(* CODESYS project TAC_Events.library
   Author: Mit Patel
   Version: 0.1.1.2
   Description: V0.1.1.0 - Initial
      V0.1.1.1 - Create RPC Sink
      V0.1.1.2 - Separate Buffer and Sink Interfaces
   Title: TAC_Events
   DefaultNamespace: TAC_Events
   Placeholder: TAC_Events
   Company: Timberline Automation and Control Co.

Project tree, tasks and I/O mapping:
  libraries: Tc2_EtherCAT, * (Beckhoff Automation GmbH); Tc2_Standard, * (Beckhoff Automation GmbH); Tc2_System, * (Beckhoff Automation GmbH); Tc2_Utilities, * (Beckhoff Automation GmbH); Tc3_JsonXml, * (Beckhoff Automation GmbH)
  ImportUtilities/
    Logger/
      data type E_LogSeverity
      function F_LogDebug [ST]
      function F_LogError [ST]
      function F_Logger [ST]
      function F_LogInfo [ST]
      function F_LogWarning [ST]
      function block FB_LogErrorEdge [ST]
      function block FB_LogInfoEdge [ST]
      function block FB_LogOnEdge [ST]
      function block FB_LogWarningEdge [ST]
      interface I_ExternalLogger: AddToLog
    String/
      Large Concats/
        function F_ClearLarge [ST]
        function F_Concat3_Large [ST]
        function F_Concat4_Large [ST]
        function F_Concat5_Large [ST]
        function F_Concat6_Large [ST]
        function F_Concat7_Large [ST]
        function F_ConcatLarge [ST]
      function F_Concat3 [ST]
      function F_Concat4 [ST]
      function F_Concat5 [ST]
      function F_Concat6 [ST]
      function F_Concat7 [ST]
      function F_StringToTarg [ST]
      function F_TargToString [ST]
      data type LongString
    global variables LogConfig
  Library/
    EventLogger/
      Bases/
        function block T_InstanceNameBase [ST]: InstanceName, SetInstanceName
      EventBuffers/
        function block T_JsonEventBuffer [ST]: FindAvailableBuffer, FindOldestBuffer, ResetBuffer, AddEvent, GetEvents, Initialise, ConvertToJson, CopyJson, EndJson, StartJson
      EventSinks/
        function block FB_CsvFileEventSink [ST]: AddEvent, GetEvents, Initialise, CyclicLogic
        function block T_RpcEventSink [ST]: AddEvent, GetEvents, Initialise
      Functions/
        function F_GetLogSeverityFromTcEventSeverity [ST]
      Interfaces/
        interface I_EventBuffer: AddEvent, GetEvents, Initialise
        interface I_EventLogger: LogEvent, ShouldLogEvent
        interface I_EventSeverityHandler: ClearLocalSeverity, GetGlobalSeverity, GetLocalSeverity, SetGlobalSeverity, SetLocalSeverity
        interface I_EventSink: AddEvent, GetEvents, Initialise
        interface I_EventSinkHandler: AddSink, ClearSinks
        interface I_Logger: LogCritical, LogError, LogInfo, LogVerbose, LogWarning
      function block T_EventLogger [ST]: LogEvent, ShouldLogEvent, ClearLocalSeverity, GetGlobalSeverity, GetLocalSeverity, SetGlobalSeverity, SetLocalSeverity, AddSink, ClearSinks, LogCritical, LogError, LogInfo, LogVerbose, LogWarning
      function block T_Logger [ST]: LogEvent, ShouldLogEvent, ClearLocalSeverity, GetGlobalSeverity, GetLocalSeverity, SetGlobalSeverity, SetLocalSeverity, LogCritical, LogError, LogInfo, LogVerbose, LogWarning, FB_init
    GVLs/
      global variables Events
      global variables EventsConfig
    Structs/
      data type ST_EventMessageBuffer
      data type ST_EventMessageBufferPool
      data type ST_EventMessageParams
      data type T_BufferString
      data type T_MessageString
    Time/
      function block FB_UnixTimestamp [ST]: TimestampMs
      interface I_TimeProvider: TimestampMs
  Project Information/
    function F_GetCompany [ST]
    function F_GetTitle [ST]
    function F_GetVersion [ST]
  Version/
    global variables Global_Version
*)

// ImportUtilities/Logger/E_LogSeverity
{attribute 'qualified_only'}
TYPE
   E_LogSeverity :
   (
      Debug := 0,
      Info := ADSLOG_MSGTYPE_HINT,
      Warning := ADSLOG_MSGTYPE_WARN,
      Error := ADSLOG_MSGTYPE_ERROR,
      None := 1000
   ) DWORD;
END_TYPE

// ImportUtilities/String/LongString
TYPE
   LongString : STRING(StringsParams.MAX_STRING_LENGTH);
END_TYPE // use StringsParams.MAX_STRING_LENGTH to adjust length

// Library/Structs/ST_EventMessageBuffer
{attribute 'pack_mode' := '0'}
TYPE ST_EventMessageBuffer :
STRUCT
 	bufferIndex : UINT := 0;
	availableForWriting : BOOL := TRUE;
  count : UINT := 0;
  timestampMs : ULINT;
  
  bufferSize : UDINT := EventsConfig.MAX_BUFFER_SIZE;
  dataSize : UDINT := 0;
END_STRUCT
END_TYPE

// Library/Structs/ST_EventMessageBufferPool
{attribute 'pack_mode' := '0'}
TYPE ST_EventMessageBufferPool :
STRUCT
  bufferCount : UINT := EventsConfig.MAX_BUFFERS;
	currentDataBufferIndex : UINT := 0;
	dataBuffers : ARRAY [1..EventsConfig.MAX_BUFFERS] OF ST_EventMessageBuffer;
END_STRUCT
END_TYPE

// Library/Structs/ST_EventMessageParams
TYPE ST_EventMessageParams :
STRUCT	
  Severity : TcEventSeverity;
  Message : T_MessageString;
  Source : T_MaxString;
END_STRUCT
END_TYPE

// Library/Structs/T_BufferString
TYPE T_BufferString : STRING(EventsConfig.MAX_BUFFER_SIZE); END_TYPE

// Library/Structs/T_MessageString
TYPE T_MessageString : STRING(EventsConfig.MAX_LOG_MESSAGE_SIZE); END_TYPE

// ImportUtilities/LogConfig
{attribute 'qualified_only'}
VAR_GLOBAL
   // set level to log. Lower log level includes higher levels i.e. info does warning and Error. 
   LogLevel : E_LogSeverity := E_LogSeverity.None; // Turn messages off by default
   ExternalLogger : I_ExternalLogger; // permit logging to something else
END_VAR

// Library/GVLs/Events
{attribute 'qualified_only'}
VAR_GLOBAL CONSTANT
  {attribute 'hide'}
  {warning disable C0228}
  _eventLogger  : T_EventLogger;                      // Global instance of event logger which will log to all sinks.
  {warning restore C0228}

  EventLogger   : I_Logger := _eventLogger;           // Global accessor for logging events.
  EventSinks    : I_EventSinkHandler := _eventLogger; // Global accessor for adding/ resetting sinks.
END_VAR

// Library/GVLs/EventsConfig
{attribute 'qualified_only'}
// Buffer Config
VAR_GLOBAL CONSTANT
  MAX_BUFFERS : UINT := 4;                    // Number of buffers.
  MAX_BUFFER_SIZE : UDINT := 65535;           // Max size in bytes of a buffer.
  CYCLE_BUFFERS : BOOL := TRUE;               // Overwrite buffers when all buffers are full.
  MAX_LOG_MESSAGE_SIZE : UINT := 512;         // Max length of log message.
  
  CSV_LOG_FILE_NAME : T_MaxString := 'logs';      // Name for CSV log files. Will have the date appended (e.g. logs_2024_05_26).
  CSV_LOG_FILE_PATH : T_MaxString := '/var/log/'; // The path for log files if using FB_CsvFileEventSink.
END_VAR

// Logs config
VAR_GLOBAL CONSTANT
  MAX_SINKS : UINT := 4; // Number of sinks.
END_VAR

// Version/Global_Version
{attribute 'TcGenerated'}
{attribute 'no-analysis'}
{attribute 'linkalways'}
// This function has been automatically generated from the project information.
VAR_GLOBAL CONSTANT
	{attribute 'const_non_replaced'}
	stLibVersion_TAC_Events : ST_LibVersion := (iMajor := 0, iMinor := 1, iBuild := 1, iRevision := 2, nFlags := 0, sVersion := '0.1.1.2');
END_VAR

// ImportUtilities/Logger/F_LogDebug
FUNCTION F_LogDebug : STRING;
VAR_INPUT
   Message : T_MaxString;
END_VAR

F_LogDebug :=
   F_Logger(
      E_LogSeverity.Debug,
      CONCAT('DEBUG ', Message)
   );

END_FUNCTION

// ImportUtilities/Logger/F_Logger
FUNCTION F_Logger : STRING;
VAR_INPUT
   LogSeverity : E_LogSeverity;
   Message : T_MaxString;
END_VAR

IF (LogSeverity < E_LogSeverity.None)
   AND_THEN (LogSeverity >= LogConfig.LogLevel) THEN

   ADSLOGSTR(LogSeverity OR ADSLOG_MSGTYPE_LOG, Message, '');
   F_Logger := Message;

   IF LogConfig.ExternalLogger <> 0 THEN
      LogConfig.ExternalLogger.AddToLog(Message, LogSeverity);
   END_IF

END_IF

END_FUNCTION

// ImportUtilities/Logger/F_LogError
FUNCTION F_LogError : STRING;
VAR_INPUT
   Message : T_MaxString;
END_VAR

F_LogError := F_Logger(ADSLOG_MSGTYPE_ERROR, Message);

END_FUNCTION

// ImportUtilities/Logger/F_LogInfo
FUNCTION F_LogInfo : STRING;
VAR_INPUT
   Message : T_MaxString;
END_VAR

F_LogInfo := F_Logger(ADSLOG_MSGTYPE_HINT, Message);

END_FUNCTION

// ImportUtilities/Logger/F_LogWarning
FUNCTION F_LogWarning : STRING;
VAR_INPUT
   Message : T_MaxString;
END_VAR

F_LogWarning := F_Logger(ADSLOG_MSGTYPE_WARN, Message);

END_FUNCTION

// ImportUtilities/Logger/FB_LogErrorEdge
FUNCTION_BLOCK FB_LogErrorEdge
VAR_INPUT
   Event : BOOL; // Event flag
   Message : T_MaxString; // Log message
   EventFallingEdge : BOOL := FALSE; // Defined which edge: FALSE = rising TRUE = falling, 
END_VAR
VAR_OUTPUT
   Q : BOOL;
END_VAR
VAR
   fbLogEdge : FB_LogOnEdge;
END_VAR

fbLogEdge(
   Event := Event,
   Message := Message,
   LogSeverity := E_LogSeverity.Error,
   EventFallingEdge := EventFallingEdge,
   Q => Q
);

END_FUNCTION_BLOCK

// ImportUtilities/Logger/FB_LogOnEdge
FUNCTION_BLOCK FB_LogOnEdge
VAR_INPUT
   Event : BOOL; // look for edge here to log.
   Message : T_MaxString; // message
   LogSeverity : E_LogSeverity; // severity
   EventFallingEdge : BOOL := FALSE; // TRUE for falling edge, FALSE for rising edge.
END_VAR
VAR_OUTPUT
   Q : BOOL;
END_VAR
VAR
   rt : R_TRIG;
   ft : F_TRIG;
END_VAR
VAR_TEMP
   logNow : BOOL;
END_VAR

rt(CLK := Event);
ft(CLK := Event);

Q := SEL(EventFallingEdge, rt.Q, ft.Q);

IF Q THEN

   CASE LogSeverity OF

      E_LogSeverity.Info:
         F_LogInfo(Message);

      E_LogSeverity.Warning:
         F_LogWarning(Message);

      E_LogSeverity.Error:
         F_LogError(Message);
   ELSE

      F_LogError(
         CONCAT(
            'Error in FB_LogOnEdge, Logseverity incorrect. Log Message for event is : ',
            Message
         )
      );

   END_CASE

END_IF

END_FUNCTION_BLOCK

// ImportUtilities/Logger/FB_LogInfoEdge
FUNCTION_BLOCK FB_LogInfoEdge
VAR_INPUT
   Event : BOOL; // Event flag
   Message : T_MaxString; // Log message
   EventFallingEdge : BOOL := FALSE; // Defined which edge: FALSE = rising TRUE = falling, 
END_VAR
VAR_OUTPUT
   Q : BOOL;
END_VAR
VAR
   fbLogEdge : FB_LogOnEdge;
END_VAR

fbLogEdge(
   Event := Event,
   Message := Message,
   LogSeverity := E_LogSeverity.Info,
   EventFallingEdge := EventFallingEdge,
   Q => Q
);

END_FUNCTION_BLOCK

// ImportUtilities/Logger/FB_LogWarningEdge
FUNCTION_BLOCK FB_LogWarningEdge
VAR_INPUT
   Event : BOOL; // Event flag
   Message : T_MaxString; // Log message
   EventFallingEdge : BOOL := FALSE; // Defined which edge: FALSE = rising TRUE = falling, 
END_VAR
VAR_OUTPUT
   Q : BOOL;
END_VAR
VAR
   fbLogEdge : FB_LogOnEdge;
END_VAR

fbLogEdge(
   Event := Event,
   Message := Message,
   LogSeverity := E_LogSeverity.Warning,
   EventFallingEdge := EventFallingEdge,
   Q => Q
);

END_FUNCTION_BLOCK

// ImportUtilities/Logger/I_ExternalLogger
INTERFACE I_ExternalLogger

METHOD AddToLog
VAR_IN_OUT
   Message : T_MaxString;
END_VAR
VAR_INPUT
   LogSeverity : E_LogSeverity;
END_VAR
END_METHOD

END_INTERFACE

// ImportUtilities/String/Large Concats/F_ClearLarge
FUNCTION F_ClearLarge
VAR_IN_OUT CONSTANT
   stringToClear : LongString;
END_VAR

MEMSET(ADR(stringToClear), 16#0, sizeof(stringToClear));

END_FUNCTION

// ImportUtilities/String/Large Concats/F_Concat3_Large
FUNCTION F_Concat3_Large : LongString;
VAR_IN_OUT CONSTANT
   StringOne : LongString;
   StringTwo : LongString;
   StringThree : LongString;
END_VAR
VAR
   str : LongString;
END_VAR

str := F_ConcatLarge(StringTwo, StringThree);

F_Concat3_Large :=
   F_ConcatLarge(
      StringOne,
      str
   );

END_FUNCTION

// ImportUtilities/String/Large Concats/F_ConcatLarge
FUNCTION F_ConcatLarge : LongString
VAR_IN_OUT CONSTANT
   StringOne : LongString;
   StringTwo : LongString;
END_VAR
VAR
   i, sizeToCpy, teminatingCharPos, maxLen : DINT;
   response : LongString;
END_VAR

maxLen := TO_DINT(StringsParams.MAX_STRING_LENGTH) - 1; // - 1 allows for terminating character in last position.

IF LEN(stringOne) + LEN(StringTwo) > maxLen THEN
   sizeToCpy := maxLen - LEN(StringTwo); //need room for the terminating character
   teminatingCharPos := maxLen; // this is the index position for utf-8 string as byte array

ELSE
   sizeToCpy := LEN(StringOne);
   teminatingCharPos := LEN(StringOne) + LEN(StringTwo);

END_IF

// copy strings into response
MEMCPY(ADR(response), ADR(StringOne), TO_UDINT(sizeToCpy));
MEMCPY(ADR(response[sizeToCpy]), ADR(StringTwo), TO_UDINT(LEN(StringTwo)));

response[teminatingCharPos] := 16#0; // string terminating character
F_ConcatLarge := response;

END_FUNCTION

// ImportUtilities/String/Large Concats/F_Concat4_Large
FUNCTION F_Concat4_Large : LongString
VAR_IN_OUT CONSTANT
   sOne : LongString;
   sTwo : LongString;
   sThree : LongString;
   sFour : LongString;
END_VAR
VAR
   str : LongString;
END_VAR

str := F_Concat3_Large(sTwo, sThree, sFour);

F_Concat4_Large :=
   F_ConcatLarge(
      sOne,
      str
   );

END_FUNCTION

// ImportUtilities/String/Large Concats/F_Concat5_Large
FUNCTION F_Concat5_Large : LongString
VAR_IN_OUT CONSTANT
   sOne : LongString;
   sTwo : LongString;
   sThree : LongString;
   sFour : LongString;
   sFive : LongString;
END_VAR
VAR
   str : LongString;
END_VAR

str := F_Concat4_Large(sTwo, sThree, sFour, sFive);
F_Concat5_Large :=
   F_ConcatLarge(
      sOne,
      str
   );

END_FUNCTION

// ImportUtilities/String/Large Concats/F_Concat6_Large
FUNCTION F_Concat6_Large : LongString
VAR_IN_OUT CONSTANT
   sOne : LongString;
   sTwo : LongString;
   sThree : LongString;
   sFour : LongString;
   sFive : LongString;
   sSix : LongString;
END_VAR
VAR
   str : LongString;
END_VAR

str := F_Concat5_Large(sTwo, sThree, sFour, sFive, sSix);
F_Concat6_Large :=
   F_ConcatLarge(
      sOne,
      str
   );

END_FUNCTION

// ImportUtilities/String/Large Concats/F_Concat7_Large
FUNCTION F_Concat7_Large : LongString
VAR_IN_OUT CONSTANT
   sOne : LongString;
   sTwo : LongString;
   sThree : LongString;
   sFour : LongString;
   sFive : LongString;
   sSix : LongString;
   sSeven : LongString;
END_VAR
VAR
   str : LongString;
END_VAR

str := F_Concat6_Large(
   sTwo,
   sThree,
   sFour,
   sFive,
   sSix,
   sSeven
);

F_Concat7_Large :=
   F_ConcatLarge(
      sOne,
      str
   );

END_FUNCTION

// ImportUtilities/String/F_Concat3
FUNCTION F_Concat3 : T_MaxString
VAR_INPUT
   StringOne : STRING;
   StringTwo : STRING;
   StringThree : STRING;
END_VAR
VAR
   response : T_MaxString;
END_VAR

response := CONCAT(StringOne, StringTwo);
response := CONCAT(response, StringThree);
F_Concat3 := response;

END_FUNCTION

// ImportUtilities/String/F_Concat4
FUNCTION F_Concat4 : T_MaxString
VAR_INPUT
   sOne : STRING;
   sTwo : STRING;
   sThree : STRING;
   sFour : STRING;
END_VAR

F_Concat4 := CONCAT(
   sOne,
   F_Concat3(sTwo, sThree, sFour)
);

END_FUNCTION

// ImportUtilities/String/F_Concat5
FUNCTION F_Concat5 : T_MaxString
VAR_INPUT
   sOne : STRING;
   sTwo : STRING;
   sThree : STRING;
   sFour : STRING;
   sFive : STRING;
END_VAR

F_Concat5 := CONCAT(
   sOne,
   F_Concat4(sTwo, sThree, sFour, sFive)
);

END_FUNCTION

// ImportUtilities/String/F_Concat6
FUNCTION F_Concat6 : T_MaxString
VAR_INPUT
   sOne : STRING;
   sTwo : STRING;
   sThree : STRING;
   sFour : STRING;
   sFive : STRING;
   sSix : STRING;
END_VAR

F_Concat6 := CONCAT(
   sOne,
   F_Concat5(sTwo, sThree, sFour, sFive, sSix)
);

END_FUNCTION

// ImportUtilities/String/F_Concat7
FUNCTION F_Concat7 : T_MaxString
VAR_INPUT
   sOne : STRING;
   sTwo : STRING;
   sThree : STRING;
   sFour : STRING;
   sFive : STRING;
   sSix : STRING;
   sSeven : STRING;
END_VAR

F_Concat7 := CONCAT(
   sOne,
   F_Concat6(
      sTwo,
      sThree,
      sFour,
      sFive,
      sSix,
      sSeven
   )
);

END_FUNCTION

// ImportUtilities/String/F_StringToTarg
FUNCTION F_StringToTarg
VAR_INPUT
   StringToConvert : T_MaxString;
END_VAR
VAR_IN_OUT
   Targ : T_ARG;
END_VAR
VAR
   b : POINTER TO BOOL;
   b8 : POINTER TO BYTE;
   w : POINTER TO WORD;
   dw : POINTER TO DWORD;
   usi : POINTER TO USINT;
   si : POINTER TO SINT;
   ui : POINTER TO UINT;
   i : POINTER TO INT;
   udi : POINTER TO UDINT;
   di : POINTER TO DINT;
   str : POINTER TO STRING;
   re : POINTER TO REAL;
   lr : POINTER TO LREAL;
END_VAR

CASE Targ.eType OF

   E_ArgType.ARGTYPE_BOOL:
      b := Targ.pData;
      b^ := TO_BOOL(StringToConvert);

   E_ArgType.ARGTYPE_BYTE:
      b8 := Targ.pData;
      b8^ := TO_BYTE(StringToConvert);

   E_ArgType.ARGTYPE_WORD:
      w := Targ.pData;
      w^ := TO_WORD(StringToConvert);

   E_ArgType.ARGTYPE_DWORD:
      dw := Targ.pData;
      dw^ := TO_DWORD(StringToConvert);

   E_ArgType.ARGTYPE_USINT:
      usi := Targ.pData;
      usi^ := TO_USINT(StringToConvert);

   E_ArgType.ARGTYPE_SINT:
      si := Targ.pData;
      si^ := TO_SINT(StringToConvert);

   E_ArgType.ARGTYPE_UINT:
      ui := Targ.pData;
      ui^ := TO_UINT(StringToConvert);

   E_ArgType.ARGTYPE_INT:
      i := Targ.pData;
      i^ := TO_INT(StringToConvert);

   E_ArgType.ARGTYPE_UDINT:
      udi := Targ.pData;
      udi^ := TO_UDINT(StringToConvert);

   E_ArgType.ARGTYPE_DINT:
      di := Targ.pData;
      di^ := TO_DINT(StringToConvert);

   E_ArgType.ARGTYPE_STRING:
      str := Targ.pData;
      str^ := TO_STRING(StringToConvert);

   E_ArgType.ARGTYPE_REAL:
      re := Targ.pData;
      re^ := TO_REAL(StringToConvert);

   E_ArgType.ARGTYPE_LREAL:
      lr := Targ.pData;
      lr^ := TO_LREAL(StringToConvert);

ELSE
   F_LogWarning(
      CONCAT(
         'Unsupported type in Targ for string conversion: ',
         TO_STRING(Targ.eType)
      )
   );
END_CASE

END_FUNCTION

// ImportUtilities/String/F_TargToString
FUNCTION F_TargToString : T_MaxString
VAR_INPUT
   Targ : T_ARG;
END_VAR
VAR
   b : POINTER TO BOOL;
   b8 : POINTER TO BYTE;
   w : POINTER TO WORD;
   dw : POINTER TO DWORD;
   usi : POINTER TO USINT;
   si : POINTER TO SINT;
   ui : POINTER TO UINT;
   i : POINTER TO INT;
   udi : POINTER TO UDINT;
   di : POINTER TO DINT;
   str : POINTER TO STRING;
   re : POINTER TO REAL;
   lr : POINTER TO LREAL;
END_VAR

CASE Targ.eType OF

   E_ArgType.ARGTYPE_BOOL:
      b := Targ.pData;
      F_TargToString := TO_STRING(b^);

   E_ArgType.ARGTYPE_BYTE:
      b8 := Targ.pData;
      F_TargToString := TO_STRING(b8^);

   E_ArgType.ARGTYPE_WORD:
      w := Targ.pData;
      F_TargToString := TO_STRING(w^);

   E_ArgType.ARGTYPE_DWORD:
      dw := Targ.pData;
      F_TargToString := TO_STRING(dw^);

   E_ArgType.ARGTYPE_USINT:
      usi := Targ.pData;
      F_TargToString := TO_STRING(usi^);

   E_ArgType.ARGTYPE_SINT:
      si := Targ.pData;
      F_TargToString := TO_STRING(si^);

   E_ArgType.ARGTYPE_UINT:
      ui := Targ.pData;
      F_TargToString := TO_STRING(ui^);

   E_ArgType.ARGTYPE_INT:
      i := Targ.pData;
      F_TargToString := TO_STRING(i^);

   E_ArgType.ARGTYPE_UDINT:
      udi := Targ.pData;
      F_TargToString := TO_STRING(udi^);

   E_ArgType.ARGTYPE_DINT:
      di := Targ.pData;
      F_TargToString := TO_STRING(di^);

   E_ArgType.ARGTYPE_STRING:
      str := Targ.pData;
      F_TargToString := TO_STRING(str^);

   E_ArgType.ARGTYPE_REAL:
      re := Targ.pData;
      F_TargToString := TO_STRING(re^);

   E_ArgType.ARGTYPE_LREAL:
      lr := Targ.pData;
      F_TargToString := TO_STRING(lr^);

ELSE
   F_LogWarning(
      CONCAT(
         'Unsupported type in Targ for string conversion: ',
         TO_STRING(Targ.eType)
      )
   );
END_CASE

END_FUNCTION

// Library/EventLogger/Bases/T_InstanceNameBase
{attribute 'reflection'} 
FUNCTION_BLOCK PUBLIC T_InstanceNameBase
VAR
  {attribute 'instance-path'} 
  {attribute 'noinit'} 
  name : T_MaxString;
  
  _instanceName : T_MaxString;
  isInstanceNameSet : BOOL := FALSE;
END_VAR

PROPERTY FINAL InstanceName : T_MaxString; // returns the fully scoped variable name
GET
IF NOT isInstanceNameSet THEN
   setInstanceName();
END_IF

InstanceName := _instanceName;
END_GET
END_PROPERTY

METHOD PRIVATE SetInstanceName
VAR
	charsToDeleteFromPath : INT;
END_VAR
//Remove Solution_Name
charsToDeleteFromPath := FIND(name, '.');
_instanceName := DELETE(name, charsToDeleteFromPath, 1);
//Remove ProjectName
charsToDeleteFromPath := FIND(_instanceName, '.');
//gives us just "FirstDeclaredPOU.etc.etc..." from above.
_instanceName := DELETE(_instanceName, charsToDeleteFromPath, 1);
END_METHOD

END_FUNCTION_BLOCK

// Library/EventLogger/EventBuffers/T_JsonEventBuffer
// Event sink which buffers log messages/ events ready for polling via RPC calls to 'GetEvents'; a method of the I_EventSink interface. 
FUNCTION_BLOCK PUBLIC T_JsonEventBuffer EXTENDS T_InstanceNameBase IMPLEMENTS I_EventBuffer
VAR
  isInitialised : BOOL := FALSE;
  
  bufferPool : ST_EventMessageBufferPool;
  jWriters : ARRAY [1..EventsConfig.MAX_BUFFERS] OF FB_JsonSaxWriter;

  _timeProvider : I_TimeProvider := NULL;
  eventId : ULINT := 0;
END_VAR

VAR CONSTANT
  NULL : UDINT := 0;
END_VAR

// Finds the first available buffer, if unable to find one and CYCLE_BUFFERS is set to TRUE, then will search for the first oldest buffer based on its timestamp.
// With CYCLE_BUFFERS set to FALSE, events will be dropped.
// Returns the buffer index from the pool, 0 (invalid) if a buffer is not found.
METHOD PRIVATE FindAvailableBuffer : UINT
VAR
  iBuffer : UINT := 0;
  iAvailable : UINT := 0;
  iOldest : UINT := 0;
END_VAR
IF NOT isInitialised THEN
  F_LogWarning(CONCAT(InstanceName, ': Unable to FindAvailableBuffer. Sink is uninitialised.'));
  RETURN;
END_IF

iAvailable := 0;

FOR iBuffer := 1 TO EventsConfig.MAX_BUFFERS DO 
  IF bufferPool.dataBuffers[iBuffer].availableForWriting THEN
    iAvailable := iBuffer;
    EXIT;
	END_IF
END_FOR

IF EventsConfig.CYCLE_BUFFERS THEN
  // All buffers are full
  IF iAvailable = 0 THEN
    iOldest := FindOldestBuffer(FALSE);
    IF iOldest > 0 AND iOldest <= EventsConfig.MAX_BUFFERS THEN
      iAvailable := iOldest;
    END_IF
  END_IF
END_IF

FindAvailableBuffer := iAvailable;
END_METHOD

// Finds the oldest buffer in the pool and returns its buffer index. Will return 0 if unable to find an old buffer.
// If checkHasItems is set to TRUE, then will only search for buffers with items, otherwise all buffers in the pool are considered.
METHOD PRIVATE FindOldestBuffer : UINT
VAR_INPUT
  checkHasItems : BOOL := FALSE;
END_VAR

VAR
  iBuffer : UINT := 0;
  iOldest : UINT := 0;
  timeOldest : ULINT;
END_VAR
IF NOT isInitialised THEN
  F_LogWarning(CONCAT(InstanceName, ': Unable to FindOldestBuffer. Sink is uninitialised.'));
  RETURN;
END_IF

IF _timeProvider = NULL THEN
  F_LogWarning(CONCAT(InstanceName, ': Unable to FindOldestBuffer. _timeProvider is uninitialised.'));
  RETURN;
END_IF

timeOldest := _timeProvider.TimestampMs;
FOR iBuffer := 1 TO EventsConfig.MAX_BUFFERS DO
  IF bufferPool.dataBuffers[iBuffer].timestampMs < timeOldest THEN
    IF NOT checkHasItems OR_ELSE bufferPool.dataBuffers[iBuffer].count > 0 THEN
      timeOldest := bufferPool.dataBuffers[iBuffer].timestampMs;
      iOldest := iBuffer;
    END_IF
  END_IF
END_FOR
    
FindOldestBuffer := iOldest;
END_METHOD

// Resets a buffer based on the input buffer index and starts the buffer ready for new events to be added.
METHOD PRIVATE ResetBuffer
VAR_INPUT
  iBuffer : UINT := 0;
END_VAR
IF NOT isInitialised THEN
  F_LogWarning(CONCAT(InstanceName, ': Unable to ResetBuffer. Sink is uninitialised.'));
  RETURN;
END_IF

IF _timeProvider = NULL THEN
  F_LogWarning(CONCAT(InstanceName, ': Unable to ResetBuffer. _timeProvider is uninitialised.'));
  RETURN;
END_IF

IF iBuffer > 0 AND iBuffer <= EventsConfig.MAX_BUFFERS THEN
  StartJson(iBuffer);
  
  bufferPool.dataBuffers[iBuffer].bufferIndex := iBuffer;
  bufferPool.dataBuffers[iBuffer].availableForWriting := TRUE;
  bufferPool.dataBuffers[iBuffer].count := 0;
  bufferPool.dataBuffers[iBuffer].bufferSize := EventsConfig.MAX_BUFFER_SIZE;
  bufferPool.dataBuffers[iBuffer].dataSize := 0;
  
  bufferPool.dataBuffers[iBuffer].timestampMs := _timeProvider.TimestampMs;
END_IF
END_METHOD

// Adds an event to the buffer for later processing.
METHOD PUBLIC AddEvent
VAR_INPUT
  eventMessageParams : ST_EventMessageParams;
END_VAR

VAR
  totalSize, messageSize : UDINT := 0;
  buffer : REFERENCE TO ST_EventMessageBuffer := 0;
END_VAR

VAR_INST
  jWriterLocal : FB_JsonSaxWriter; // For calculating message size.
END_VAR

VAR CONSTANT
  END_JSON_ARRAY_SIZE : UINT := 3; // End array, end object and null terminator.
END_VAR
IF NOT isInitialised THEN
  F_LogWarning(CONCAT(InstanceName, ': Unable to AddEvent. Sink is uninitialised.'));
  RETURN;
END_IF

jWriterLocal.ResetDocument();
messageSize := ConvertToJson(eventMessageParams, jWriter := jWriterLocal);

IF bufferPool.currentDataBufferIndex = 0 OR bufferPool.currentDataBufferIndex > EventsConfig.MAX_BUFFERS THEN // Try to find an empty buffer.
	bufferPool.currentDataBufferIndex := FindAvailableBuffer();
  ResetBuffer(bufferPool.currentDataBufferIndex);
END_IF

IF bufferPool.currentDataBufferIndex > 0 AND bufferPool.currentDataBufferIndex <= EventsConfig.MAX_BUFFERS THEN 
  buffer REF= bufferPool.dataBuffers[bufferPool.currentDataBufferIndex];

  IF buffer.dataSize + messageSize > (EventsConfig.MAX_BUFFER_SIZE - END_JSON_ARRAY_SIZE) THEN  // Will adding this event cause the buffer to overflow?
    EndJson(bufferPool.currentDataBufferIndex);
    buffer.availableForWriting := FALSE; // Available for reading/ sending

	  bufferPool.currentDataBufferIndex := FindAvailableBuffer(); // Next buffer for writing. Will return 0 if no available buffers.
    ResetBuffer(bufferPool.currentDataBufferIndex);
  END_IF
END_IF

IF bufferPool.currentDataBufferIndex > 0 AND bufferPool.currentDataBufferIndex <= EventsConfig.MAX_BUFFERS THEN // Check bounds again due to buffer index change above.
  buffer REF= bufferPool.dataBuffers[bufferPool.currentDataBufferIndex]; // Buffer index has changed so update the internal ref.
  IF buffer.availableForWriting THEN
    ConvertToJson(eventMessageParams, jWriter := jWriters[bufferPool.currentDataBufferIndex]);
    totalSize := jWriters[bufferPool.currentDataBufferIndex].GetDocumentLength();                 
    buffer.dataSize := totalSize;
    buffer.count := buffer.count + 1;
    eventId := eventId + 1;
  END_IF
END_IF
END_METHOD

// Gets events currently stored in the buffer and copies them to the resultString, returning the total length of bytes copied.
METHOD PUBLIC GetEvents : UDINT
VAR_INPUT
  resultString : REFERENCE TO T_BufferString;
END_VAR

VAR
  iBuffer : UINT := 0;
  totalSize : UDINT := 0;
END_VAR

VAR CONSTANT
  // Note that the size returned from any 
  // json writer's GetDocumentLength method 
  // includes the null terminator, which we want to remove.
  // This is due to the JSON parsers in .NET or Influx's Telegraf, etc
  // not being able to understand the null terminator and throwing errors,
  // e.g. stating that there are additional characters at the end of the JSON payload.
  REMOVE_NULL_TERMINATOR : UDINT := 1;
END_VAR
IF NOT isInitialised THEN
  F_LogWarning(CONCAT(InstanceName, ': Unable to GetEvents. Sink is uninitialised.'));
  RETURN;
END_IF

iBuffer := FindOldestBuffer(TRUE);
IF iBuffer > 0 AND iBuffer <= EventsConfig.MAX_BUFFERS THEN
  IF NOT bufferPool.dataBuffers[iBuffer].availableForWriting THEN
    IF bufferPool.dataBuffers[iBuffer].count > 0 THEN
      totalSize := CopyJson(iBuffer, resultString);
      ResetBuffer(iBuffer);
    END_IF
  ELSE // Current buffer
    IF bufferPool.dataBuffers[iBuffer].count > 0 THEN
      bufferPool.dataBuffers[iBuffer].availableForWriting := FALSE; // Available for reading/ sending
      EndJson(iBuffer);
      totalSize := CopyJson(iBuffer, resultString);
      ResetBuffer(iBuffer);
      bufferPool.currentDataBufferIndex := FindAvailableBuffer(); // Next buffer for writing. Will return 0 if no available buffers.
      ResetBuffer(bufferPool.currentDataBufferIndex);
    END_IF
  END_IF
END_IF

GetEvents := totalSize - REMOVE_NULL_TERMINATOR;
END_METHOD

// Initialises the buffer including an I_TimeProvider for timestamping buffers and events.
METHOD PUBLIC Initialise
VAR_INPUT
	timeProvider : I_TimeProvider;
END_VAR

VAR
  iBuffer : UINT := 0;
END_VAR
_timeProvider := timeProvider;

IF _timeProvider = NULL THEN
  F_LogWarning(CONCAT(InstanceName, ': Unable to Initialise. _timeProvider is uninitialised.'));
  RETURN;
END_IF

isInitialised := TRUE;

FOR iBuffer := 1 TO EventsConfig.MAX_BUFFERS DO 
  ResetBuffer(iBuffer);
END_FOR
END_METHOD

// Converts the input eventMessageParams to JSON (without string copying).
METHOD PRIVATE ConvertToJson
VAR_INPUT
  eventMessageParams : ST_EventMessageParams;
END_VAR

VAR_OUTPUT
  docSize : UDINT;
END_VAR

VAR_IN_OUT
  jWriter : FB_JsonSaxWriter;
END_VAR

VAR
  timestampMs : ULINT;
  severity : T_MaxString;
END_VAR
IF NOT isInitialised THEN
  F_LogWarning(CONCAT(InstanceName, ': Unable to ConvertToJson. Sink is uninitialised.'));
  RETURN;
END_IF

IF _timeProvider = NULL THEN
  F_LogWarning(CONCAT(InstanceName, ': Unable to ConvertToJson. _timeProvider is uninitialised.'));
  RETURN;
END_IF

timestampMs := _timeProvider.TimestampMs;
severity := TO_STRING(eventMessageParams.Severity);

jWriter.StartObject();

  jWriter.AddKey('EventId');
  jWriter.AddUlint(eventId);

  jWriter.AddKeyString('Severity', severity);
  jWriter.AddKey('FileTime'); // Add unix timestamp
  jWriter.AddUlint(timestampMs);
  jWriter.AddKeyString('SourceName', eventMessageParams.Source); 
  jWriter.AddKeyString('MessageBody', eventMessageParams.Message);
  
jWriter.EndObject();

docSize := jWriter.GetDocumentLength();
END_METHOD

// Copies data in the JSON writer and returns the total length of bytes copied.
METHOD PRIVATE CopyJson : UDINT
VAR_INPUT
  iBuffer : UINT := 0;
  resultString : REFERENCE TO T_BufferString;
END_VAR

VAR
  totalSize : UDINT := 0;
END_VAR

VAR CONSTANT
  RESULT_STRING_SIZE : UDINT := SIZEOF(resultString);
END_VAR
IF NOT isInitialised THEN
  F_LogWarning(CONCAT(InstanceName, ': Unable to CopyJson. Sink is uninitialised.'));
  RETURN;
END_IF

IF iBuffer = 0 OR iBuffer > EventsConfig.MAX_BUFFERS THEN
	RETURN;
END_IF

MEMSET(ADR(resultString), 0, RESULT_STRING_SIZE); // Copy doc should overwrite resultString including null termination characters. 

totalSize := jWriters[iBuffer].CopyDocument
             (
               PDoc := resultString, 
               nDoc := RESULT_STRING_SIZE
             );
             
bufferPool.dataBuffers[iBuffer].dataSize := totalSize;
CopyJson := totalSize;
END_METHOD

// Ends the JSON string, ready for the JSON string to be copied.
METHOD PRIVATE EndJson
VAR_INPUT
  iBuffer : UINT := 0;
END_VAR
IF NOT isInitialised THEN
  F_LogWarning(CONCAT(InstanceName, ': Unable to EndJson. Sink is uninitialised.'));
  RETURN;
END_IF

IF iBuffer = 0 OR iBuffer > EventsConfig.MAX_BUFFERS THEN
	RETURN;
END_IF

jWriters[iBuffer].EndArray();
jWriters[iBuffer].EndObject();
END_METHOD

// Starts the JSON string, for additional JSON objects can be appended.
METHOD PRIVATE StartJson
VAR_INPUT
  iBuffer : UINT := 0;
END_VAR
IF NOT isInitialised THEN
  F_LogWarning(CONCAT(InstanceName, ': Unable to StartJson. Sink is uninitialised.'));
  RETURN;
END_IF

IF iBuffer = 0 OR iBuffer > EventsConfig.MAX_BUFFERS THEN
	RETURN;
END_IF

jWriters[iBuffer].ResetDocument();  
jWriters[iBuffer].StartObject();
jWriters[iBuffer].AddKey('Logs');
jWriters[iBuffer].StartArray();
END_METHOD

END_FUNCTION_BLOCK

// Library/EventLogger/Interfaces/I_EventSink
// Interface for consuming and exposing event logs for transmitting to an event receiver/ listener.
INTERFACE I_EventSink

// Adds an event to the sink for processing.
METHOD AddEvent
VAR_INPUT
  eventMessageParams : ST_EventMessageParams;
END_VAR
END_METHOD

// Gets events currently stored in the buffer and copies them to the resultString.
METHOD GetEvents : T_BufferString;
END_METHOD

// Initialises the sink including an I_TimeProvider for timestamping events.
METHOD Initialise
VAR_INPUT
	timeProvider : I_TimeProvider;
END_VAR
END_METHOD

END_INTERFACE

// Library/Time/I_TimeProvider
INTERFACE I_TimeProvider

PROPERTY TimestampMs : ULINT
GET
END_GET
END_PROPERTY

END_INTERFACE

// Library/EventLogger/Interfaces/I_EventBuffer
// Interface for buffering event logs.
INTERFACE I_EventBuffer

// Adds an event to the buffer for later processing.
METHOD AddEvent
VAR_INPUT
  eventMessageParams : ST_EventMessageParams;
END_VAR
END_METHOD

// Gets events currently stored in the buffer and copies them to the resultString, returning the total length of bytes copied.
METHOD GetEvents : UDINT
VAR_INPUT
  resultString : REFERENCE TO T_BufferString;
END_VAR
END_METHOD

// Initialises the buffer including an I_TimeProvider for timestamping buffers and events.
METHOD Initialise
VAR_INPUT
	timeProvider : I_TimeProvider;
END_VAR
END_METHOD

END_INTERFACE

// Library/EventLogger/EventSinks/FB_CsvFileEventSink
// Event sink which writes log messages/ events to a CSV file. 
FUNCTION_BLOCK PUBLIC FB_CsvFileEventSink EXTENDS T_InstanceNameBase IMPLEMENTS I_EventSink
VAR
  isInitialised : BOOL := FALSE;
  
  csvFileWriter : T_CsvFileWriter;
  
  _timeProvider : I_TimeProvider := NULL;
  
  // Timeout timer to write messages in the T_CsvFileWriter's buffer after a timeout period.
  timeoutDuration : TIME := T#2S;         
  startTimer : BOOL := TRUE;
  timeoutTrigger : TON := (IN := startTimer, PT := timeoutDuration);
  
  task : T_Task;
  currentDateTime : T_MaxString;
  eventId : ULINT := 0;
END_VAR

VAR CONSTANT
  NULL : UDINT := 0;
END_VAR

// Adds an event to the sink for processing.
METHOD PUBLIC AddEvent
VAR_INPUT
  eventMessageParams : ST_EventMessageParams;
END_VAR
IF NOT isInitialised THEN
  F_LogWarning(CONCAT(InstanceName, ': Unable to AddEvent. Sink is uninitialised.'));
  RETURN;
END_IF

IF task.DateString <> currentDateTime THEN
  currentDateTime := task.DateString;
  csvFileWriter.SetFileParams(F_Concat3(EventsConfig.CSV_LOG_FILE_PATH, F_Concat3(EventsConfig.CSV_LOG_FILE_NAME, '_', currentDateTime), '.csv'), ASCI_COMMA);
END_IF

csvFileWriter.AddStringField(TO_STRING(eventId));
csvFileWriter.AddStringField(TO_STRING(_timeProvider.TimestampMs));
csvFileWriter.AddStringField(TO_STRING(eventMessageParams.Severity));
csvFileWriter.AddStringField(eventMessageParams.Source);
csvFileWriter.AddStringField(eventMessageParams.Message);

// Todo. Additional fields, unix timestamp, event id etc.

csvFileWriter.NewLine();
eventId := eventId + 1;
END_METHOD

// Gets events currently stored in the buffer and copies them to the resultString.
METHOD PUBLIC GetEvents : T_BufferString;
IF NOT isInitialised THEN
  F_LogWarning(CONCAT(InstanceName, ': Unable to GetEvents. Sink is uninitialised.'));
  RETURN;
END_IF

csvFileWriter.WriteToFile();
END_METHOD

// Initialises the buffer including an I_TimeProvider for timestamping buffers and events.
METHOD PUBLIC Initialise
VAR_INPUT
	timeProvider : I_TimeProvider;
END_VAR
_timeProvider := timeProvider;

IF _timeProvider = NULL THEN
  F_LogWarning(CONCAT(InstanceName, ': Unable to Initialise. _timeProvider is uninitialised.'));
  RETURN;
END_IF

isInitialised := TRUE;

currentDateTime := task.DateString;
csvFileWriter.SetFileOpenMode(TRUE);
csvFileWriter.SetFileParams(F_Concat3(EventsConfig.CSV_LOG_FILE_PATH, F_Concat3(EventsConfig.CSV_LOG_FILE_NAME, '_', currentDateTime), '.csv'), ASCI_COMMA);
END_METHOD

METHOD PUBLIC CyclicLogic
IF NOT isInitialised THEN
  F_LogWarning(CONCAT(InstanceName, ': Unable to Execute. Sink is uninitialised.'));
  RETURN;
END_IF

csvFileWriter();

timeoutTrigger(IN := startTimer); // Restart timer on next cycle if triggered
IF timeoutTrigger.Q THEN
  timeoutTrigger(IN := FALSE);
  GetEvents();                    // Write data in the buffer.
END_IF
END_METHOD

END_FUNCTION_BLOCK

// Library/EventLogger/EventSinks/T_RpcEventSink
// Event sink which buffers log messages/ events ready for polling via RPC calls to 'GetEvents'; a method of the I_EventSink interface. 
FUNCTION_BLOCK PUBLIC T_RpcEventSink EXTENDS T_InstanceNameBase IMPLEMENTS I_EventSink
VAR
  jsonBuffer : T_JsonEventBuffer;
END_VAR

// Adds an event to the sink for processing.
METHOD PUBLIC AddEvent
VAR_INPUT
  eventMessageParams : ST_EventMessageParams;
END_VAR
jsonBuffer.AddEvent(eventMessageParams);
END_METHOD

// Gets events currently stored in the buffer and copies them to the resultString.
{attribute 'TcRpcEnable'}
METHOD PUBLIC GetEvents : T_BufferString;
jsonBuffer.GetEvents(GetEvents);
END_METHOD

// Initialises the buffer including an I_TimeProvider for timestamping buffers and events.
METHOD PUBLIC Initialise
VAR_INPUT
	timeProvider : I_TimeProvider;
END_VAR
jsonBuffer.Initialise(timeProvider);
END_METHOD

END_FUNCTION_BLOCK

// Library/EventLogger/Functions/F_GetLogSeverityFromTcEventSeverity
// Conversion helper to convert from TcEventSeverity to Intecre.Utilities E_LogSeverity.
FUNCTION INTERNAL F_GetLogSeverityFromTcEventSeverity : E_LogSeverity
VAR_INPUT
  severity : TcEventSeverity;
END_VAR

CASE severity OF

  TcEventSeverity.Verbose   : F_GetLogSeverityFromTcEventSeverity := E_LogSeverity.Debug;
  TcEventSeverity.Info      : F_GetLogSeverityFromTcEventSeverity := E_Logseverity.Info;
  TcEventSeverity.Warning   : F_GetLogSeverityFromTcEventSeverity := E_Logseverity.Warning;
  TcEventSeverity.Error     : F_GetLogSeverityFromTcEventSeverity := E_Logseverity.Error;
  TcEventSeverity.Critical  : F_GetLogSeverityFromTcEventSeverity := E_Logseverity.Error;

END_CASE

END_FUNCTION

// Library/EventLogger/Interfaces/I_EventLogger
// Internal interface for general logging methods required by all loggers.
INTERFACE INTERNAL I_EventLogger

// Generic logging method.
METHOD INTERNAL LogEvent
VAR_IN_OUT CONSTANT
  message : T_MessageString; 
  sourceInstanceName : T_MaxString;
END_VAR

VAR_INPUT
  severity : TcEventSeverity;
END_VAR
END_METHOD

// Checks severity filters for whether the log message/ event should be logged.
METHOD INTERNAL ShouldLogEvent : BOOL
VAR_INPUT
  severity : TcEventSeverity;
END_VAR
END_METHOD

END_INTERFACE

// Library/EventLogger/Interfaces/I_EventSeverityHandler
// Interface for setting/ clearing local severity level.
INTERFACE I_EventSeverityHandler

// Clear the currently set local severity level.
METHOD ClearLocalSeverity
END_METHOD

// Get global severity level.
METHOD GetGlobalSeverity : TcEventSeverity
END_METHOD

// Get local severity level.
METHOD GetLocalSeverity : TcEventSeverity
END_METHOD

// Set a global severity level to filter logged events.
METHOD SetGlobalSeverity
VAR_INPUT
  severity : TcEventSeverity;
END_VAR
END_METHOD

// Set a local severity level to filter logged events. Ensure clear is called once local logging is complete.
METHOD SetLocalSeverity
VAR_INPUT
  severity : TcEventSeverity;
END_VAR
END_METHOD

END_INTERFACE

// Library/EventLogger/Interfaces/I_EventSinkHandler
// Interface for handling sinks. Allows adding/ clearing sinks to be processed.
INTERFACE I_EventSinkHandler

// Adds a sink to the sink handler and returns TRUE if successful.
METHOD AddSink : BOOL
VAR_INPUT	
  sink : I_EventSink;
END_VAR
END_METHOD

// Clears all sinks currently being handled by the sink handler.
METHOD ClearSinks
END_METHOD

END_INTERFACE

// Library/EventLogger/Interfaces/I_Logger
// Interface for logging methods which can be called in user code.
INTERFACE I_Logger

METHOD LogCritical
VAR_INPUT
  message : T_MessageString; 
END_VAR
END_METHOD

METHOD LogError
VAR_INPUT
  message : T_MessageString; 
END_VAR
END_METHOD

METHOD LogInfo
VAR_INPUT
  message : T_MessageString; 
END_VAR
END_METHOD

METHOD LogVerbose
VAR_INPUT
  message : T_MessageString; 
END_VAR
END_METHOD

METHOD LogWarning
VAR_INPUT
  message : T_MessageString; 
END_VAR
END_METHOD

END_INTERFACE

// Library/EventLogger/T_EventLogger
// Internal logger which allows adding/ clearing sinks to be processed, in addition to receiving log events and forwarding them to sinks.
FUNCTION_BLOCK INTERNAL T_EventLogger EXTENDS T_InstanceNameBase IMPLEMENTS I_EventLogger, I_Logger, I_EventSinkHandler, I_EventSeverityHandler;
VAR
  eventSinks : ARRAY[1..EventsConfig.MAX_SINKS] OF I_EventSink;
  eventSinksCount : UINT := 0;
  
  globalSeverity : TcEventSeverity; // Global log filter.
  localSeverity : TcEventSeverity;
  useLocalSeverity : BOOL;
END_VAR

VAR CONSTANT
  NULL : UDINT := 0;
END_VAR

METHOD INTERNAL LogEvent
VAR_IN_OUT CONSTANT
  message : T_MessageString; 
  sourceInstanceName : T_MaxString;
END_VAR

VAR_INPUT
  severity : TcEventSeverity;
END_VAR

VAR
  iSink : UINT := 0;
  adsLogSeverity : E_LogSeverity;
  eventMessageParams : ST_EventMessageParams;
END_VAR
IF NOT ShouldLogEvent(severity) THEN
  RETURN;
END_IF

eventMessageParams.Message := message;
eventMessageParams.Severity := severity;
eventMessageParams.Source := sourceInstanceName;

IF eventSinksCount > 0 AND eventSinksCount <= EventsConfig.MAX_SINKS THEN
  FOR iSink := 1 TO eventSinksCount DO
    IF eventSinks[iSink] <> NULL THEN
      eventSinks[iSink].AddEvent(eventMessageParams);
    ELSE
      F_LogWarning(CONCAT(InstanceName, ': Unable to LogEvent. Sink is uninitialised.'));
    END_IF
  END_FOR
END_IF

adsLogSeverity := F_GetLogSeverityFromTcEventSeverity(severity);
F_Logger(
  LogSeverity := adsLogSeverity,
  Message := F_Concat3(sourceInstanceName, ': ', message)
);
END_METHOD

METHOD INTERNAL ShouldLogEvent : BOOL
VAR_INPUT
  severity : TcEventSeverity;
END_VAR
IF useLocalSeverity THEN
  ShouldLogEvent := severity >= localSeverity;  
ELSE
  ShouldLogEvent := severity >= globalSeverity;
END_IF
END_METHOD

// Clear the currently set local severity level.
METHOD PUBLIC ClearLocalSeverity
useLocalSeverity := FALSE;
END_METHOD

// Get global severity level.
METHOD GetGlobalSeverity : TcEventSeverity
GetGlobalSeverity := globalSeverity;
END_METHOD

// Get local severity level.
METHOD GetLocalSeverity : TcEventSeverity
GetLocalSeverity := localSeverity;
END_METHOD

// Set a global severity level to filter logged events.
METHOD PUBLIC SetGlobalSeverity
VAR_INPUT
	severity	: TcEventSeverity;
END_VAR
globalSeverity := severity;
END_METHOD

// Set a local severity level to filter logged events. Ensure clear is called once local logging is complete.
METHOD PUBLIC SetLocalSeverity
VAR_INPUT
	severity	: TcEventSeverity;
END_VAR
localSeverity := severity;
useLocalSeverity := TRUE;
END_METHOD

// Adds a sink to the sink handler and returns TRUE if successful.
METHOD PUBLIC AddSink : BOOL
VAR_INPUT
	sink	: I_EventSink;
END_VAR
IF eventSinksCount + 1 > EventsConfig.MAX_SINKS THEN
  F_LogWarning(CONCAT(InstanceName, ': Unable to add sink. Maximum number of event sinks reached'));
  RETURN;
END_IF

eventSinksCount := eventSinksCount + 1;
eventSinks[eventSinksCount] := sink;
AddSink := TRUE;
END_METHOD

// Clears all sinks currently being handled by the sink handler.
METHOD PUBLIC ClearSinks
VAR
  iSink : UINT := 0;
END_VAR
IF eventSinksCount > 0 AND eventSinksCount <= EventsConfig.MAX_SINKS THEN
  FOR iSink := 1 TO eventSinksCount DO
    eventSinks[iSink] := NULL;
  END_FOR
END_IF

eventSinksCount := 0;
END_METHOD

METHOD PUBLIC LogCritical
VAR_INPUT
  message : T_MessageString; 
END_VAR

VAR
  localInstanceName : T_MaxString;
END_VAR
localInstanceName := InstanceName;
LogEvent(message := message, sourceInstanceName := localInstanceName, severity := TcEventSeverity.Critical);
END_METHOD

METHOD PUBLIC LogError
VAR_INPUT
  message : T_MessageString; 
END_VAR

VAR
  localInstanceName : T_MaxString;
END_VAR
localInstanceName := InstanceName;
LogEvent(message := message, sourceInstanceName := localInstanceName, severity := TcEventSeverity.Error);
END_METHOD

METHOD PUBLIC LogInfo
VAR_INPUT
  message : T_MessageString; 
END_VAR

VAR
  localInstanceName : T_MaxString;
END_VAR
localInstanceName := InstanceName;
LogEvent(message := message, sourceInstanceName := localInstanceName, severity := TcEventSeverity.Info);
END_METHOD

METHOD PUBLIC LogVerbose
VAR_INPUT
  message : T_MessageString; 
END_VAR

VAR
  localInstanceName : T_MaxString;
END_VAR
localInstanceName := InstanceName;
LogEvent(message := message, sourceInstanceName := localInstanceName, severity := TcEventSeverity.Verbose);
END_METHOD

METHOD PUBLIC LogWarning
VAR_INPUT
  message : T_MessageString; 
END_VAR

VAR
  localInstanceName : T_MaxString;
END_VAR
localInstanceName := InstanceName;
LogEvent(message := message, sourceInstanceName := localInstanceName, severity := TcEventSeverity.Warning);
END_METHOD

END_FUNCTION_BLOCK

// Library/EventLogger/T_Logger
// Logger for allowing events of any level to be raised in addition to being able to set/clear a local severity for specific logs.
FUNCTION_BLOCK PUBLIC T_Logger EXTENDS T_InstanceNameBase IMPLEMENTS I_EventLogger, I_Logger, I_EventSeverityHandler
VAR CONSTANT
  NULL : UDINT := 0;
END_VAR

METHOD INTERNAL LogEvent
VAR_IN_OUT CONSTANT
  message : T_MessageString; 
  sourceInstanceName : T_MaxString;
END_VAR

VAR_INPUT
  severity : TcEventSeverity;
END_VAR
IF Events.EventLogger = NULL THEN
  F_LogWarning(CONCAT(InstanceName, ': Unable to LogEvent. Events.EventLogger is null/ uninitialised.'));
  RETURN;
END_IF

IF NOT ShouldLogEvent(severity) THEN
  RETURN;
END_IF

Events._eventLogger.LogEvent(
    message:= message, 
    sourceInstanceName:= sourceInstanceName, 
    severity:= severity
  );
END_METHOD

METHOD INTERNAL ShouldLogEvent : BOOL
VAR_INPUT
  severity : TcEventSeverity;
END_VAR
ShouldLogEvent := TRUE;
END_METHOD

// Clear the currently set local severity level.
METHOD PUBLIC ClearLocalSeverity
Events._eventLogger.ClearLocalSeverity();
END_METHOD

// Get global severity level.
METHOD GetGlobalSeverity : TcEventSeverity
GetGlobalSeverity := Events._eventLogger.GetGlobalSeverity();
END_METHOD

// Get local severity level.
METHOD GetLocalSeverity : TcEventSeverity
GetLocalSeverity := Events._eventLogger.GetLocalSeverity();
END_METHOD

// Set a global severity level to filter logged events.
METHOD PUBLIC SetGlobalSeverity
VAR_INPUT
	severity	: TcEventSeverity;
END_VAR
Events._eventLogger.SetGlobalSeverity(severity);
END_METHOD

// Set a local severity level to filter logged events. Ensure clear is called once local logging is complete.
METHOD PUBLIC SetLocalSeverity
VAR_INPUT
	severity	: TcEventSeverity;
END_VAR
Events._eventLogger.SetLocalSeverity(severity);
END_METHOD

METHOD PUBLIC LogCritical
VAR_INPUT
	message	: T_MessageString;
END_VAR

VAR
  localInstanceName : T_MaxString;
END_VAR
localInstanceName := InstanceName;
LogEvent(message := message, sourceInstanceName := localInstanceName, severity := TcEventSeverity.Critical);;
END_METHOD

METHOD PUBLIC LogError
VAR_INPUT
	message	: T_MessageString;
END_VAR

VAR
  localInstanceName : T_MaxString;
END_VAR
localInstanceName := InstanceName;
LogEvent(message := message, sourceInstanceName := localInstanceName, severity := TcEventSeverity.Error);
END_METHOD

METHOD PUBLIC LogInfo
VAR_INPUT
	message	: T_MessageString;
END_VAR

VAR
  localInstanceName : T_MaxString;
END_VAR
localInstanceName := InstanceName;
LogEvent(message := message, sourceInstanceName := localInstanceName, severity := TcEventSeverity.Info);
END_METHOD

METHOD PUBLIC LogVerbose
VAR_INPUT
	message	: T_MessageString;
END_VAR

VAR
  localInstanceName : T_MaxString;
END_VAR
localInstanceName := InstanceName;
LogEvent(message := message, sourceInstanceName := localInstanceName, severity := TcEventSeverity.Verbose);
END_METHOD

METHOD PUBLIC LogWarning
VAR_INPUT
	message	: T_MessageString;
END_VAR

VAR
  localInstanceName : T_MaxString;
END_VAR
localInstanceName := InstanceName;
LogEvent(message := message, sourceInstanceName := localInstanceName, severity := TcEventSeverity.Warning);
END_METHOD

{attribute 'hide'}
METHOD FB_init : BOOL
VAR_INPUT
	bInitRetains : BOOL; // if TRUE, the retain variables are initialized (warm start / cold start)
	bInCopyCode : BOOL;  // if TRUE, the instance afterwards gets moved into the copy code (online change)
END_VAR
// Ensure Intecre_Utilities log level is set to Debug so all logs are processed. 
// Log filtering is handled via Events.GLOBAL_LOG_SEVERITY and I_Logger -> I_EventSeverityHandler for setting local severity.
// See events tester.
//Intecre_Utilities.LogConfig.LogLevel := E_LogSeverity.Debug; 

// Set the minimum global logging severity to filter all events.
SetGlobalSeverity(TcEventSeverity.Verbose);
END_METHOD

END_FUNCTION_BLOCK

// Library/Time/FB_UnixTimestamp
// Timestamp provider for calculating Unix time. Required to be called in a cyclic manner.
FUNCTION_BLOCK PUBLIC FB_UnixTimestamp IMPLEMENTS I_TimeProvider
VAR_OUTPUT
	milliseconds : ULINT;
	cpuMicroSeconds : ULINT;
	systemMicroSeconds : ULINT;
	dcToTimeZoneMicroSeconds : ULINT;
END_VAR

VAR
	localSystemTime : FB_LocalSystemTime := (bEnable := TRUE, dwCycle := 1);
	getTimeZoneInformation : FB_GetTimeZoneInformation;
	timeZoneInformation : ST_TimeZoneInformation;
	specificLocalTimeToFileTime, specificDcToFileTime : FB_TzSpecificLocalTimeToFileTime;
	fileTime, dcFileTime, dcToFileTime : T_FILETIME;
	onZerothSecondLastCycle : BOOL;
	tDcTime : T_DCTIME64;

	cpuHighTime, systemHighTime : UDINT;
	cpuLowTime, systemLowTime : UDINT;
	getSystemTime : GETSYSTEMTIME;
	getCPUCounter : GETCPUCOUNTER;
	diffBetweenSystemAndDc, prevDiff : ULINT;
  _timestampMs : ULINT;
END_VAR

// Get local system time
tDcTime := F_GetCurDcTaskTime64();
localSystemTime();
getCPUCounter( cpuCntHiDW => cpuHighTime, cpuCntLoDW => cpuLowTime );
getSystemTime( timeHiDW => systemHighTime, timeLoDW => systemLowTime );

// On the zeroth second of each minutesync timezone information
IF (timeZoneInformation.standardName = '' OR (localSystemTime.systemTime.wSecond = 0 AND NOT onZerothSecondLastCycle)) THEN
	getTimeZoneInformation( sNetID := '', bExecute := TRUE, tzInfo => timeZoneInformation );
END_IF;

// Convert local system time to unix timestamps
specificLocalTimeToFileTime(
		in := Tc2_Utilities.SYSTEMTIME_TO_FILETIME( localSystemTime.systemTime ),
		tzInfo := timeZoneInformation,
		out => fileTime
	);

_timestampMs := milliseconds := (SHL( DWORD_TO_ULINT( fileTime.dwHighDateTime ), 32 ) + DWORD_TO_ULINT( fileTime.dwLowDateTime )) / 10000 - 11644473600000;

onZerothSecondLastCycle := localSystemTime.systemTime.wSecond = 0;

specificDcToFileTime( in := DCTIME64_TO_FILETIME( tDcTime ), tzInfo := timeZoneInformation, out => dcFileTime );
dcToTimeZoneMicroSeconds :=
	(SHL( DWORD_TO_ULINT( dcFileTime.dwHighDateTime ), 32 ) + DWORD_TO_ULINT( dcFileTime.dwLowDateTime )) / 10 - 11644473600000000;

cpuMicroSeconds := (SHL( DWORD_TO_ULINT( cpuHighTime ), 32 ) + DWORD_TO_ULINT( cpuLowTime )) / 10 - 11644473600000000;
systemMicroSeconds := (SHL( DWORD_TO_ULINT( systemHighTime ), 32 ) + DWORD_TO_ULINT( systemLowTime )) / 10 - 11644473600000000;

//diffBetweenSystemAndDc := dcToTimeZoneMilliSeconds - localSysTimeMlSec;

PROPERTY TimestampMs : ULINT
GET
TimestampMs := milliseconds;
END_GET
END_PROPERTY

END_FUNCTION_BLOCK

// Project Information/F_GetCompany
// This function has been automatically generated from the project information.
{attribute 'signature_flag' := '1073741824'}
{attribute 'TcGenerated'}
{attribute 'no-analysis'}
FUNCTION F_GetCompany : WSTRING
VAR_INPUT
	
END_VAR

F_GetCompany := "Timberline Automation and Control Co.";

END_FUNCTION

// Project Information/F_GetTitle
// This function has been automatically generated from the project information.
{attribute 'signature_flag' := '1073741824'}
{attribute 'TcGenerated'}
{attribute 'no-analysis'}
FUNCTION F_GetTitle : WSTRING
VAR_INPUT
	
END_VAR

F_GetTitle := "TAC_Events";

END_FUNCTION

// Project Information/F_GetVersion
// This function has been automatically generated from the project information.
{attribute 'signature_flag' := '1073741824'}
{attribute 'TcGenerated'}
{attribute 'no-analysis'}
FUNCTION F_GetVersion : ST_LibVersion
VAR_INPUT
	
END_VAR

F_GetVersion.iMajor := 0;
F_GetVersion.iMinor := 1;
F_GetVersion.iBuild := 1;
F_GetVersion.iRevision := 2;
F_GetVersion.sVersion := '0.1.1.2';
F_GetVersion.nFlags := 0;

END_FUNCTION
